KUKA KRL program: vw_bu_usr_s.src, vw_bu_usr_s.dat

--- vw_bu_usr_s.src ---
&ACCESS RV1
&COMMENT KS26
&REL 200
&PARAM DISKPATH = VW_User/Applikation/BU_Buersten
&PARAM TPUSER_VERSION = 8.3.0
DEF VW_BU_USR_S( )
;
;***************************************************
;*Technologiepaket Buersten                        *
;*                                                 *
;*Konzernstandard                                  *
;*Bearbeiter: C. Eisenknappl AUDI AG I/PG-C61      *
;*                                                 *
;* Aenderungsjournal:                              *
;*                                                 *
;***************************************************
;
END
;
;FOLD INIT BU
GLOBAL DEF BU_INIT( )
INT i
;
;FOLD Version Techpaket
Tech_BU.Name[]="KS26.01.002_20190612"
;ENDFOLD
;
;FOLD Vorbesetzung Meldungsausgabe
FOR i=1 TO 100
  n_BUS_Handle[i]=-1
  n_BUR_Handle[i]=-1
ENDFOR
;ENDFOLD
;
;FOLD BU BASE ADRESSEN INITIALISIEREN
BU_BASE_INIT( )
;ENDFOLD
;
END
;ENDFOLD
;
;***************************************************
;FOLD SAW BU
GLOBAL DEF BU_SAW( )
INT i
;
;
END
;ENDFOLD
;
;***************************************************
;FOLD RESET BU
GLOBAL DEF BU_RESET( )
INT i
;
;
END
;ENDFOLD
;
;***************************************************
;FOLD CANCEL BU
GLOBAL DEF BU_CANCEL( )
INT i
;
;
END
;ENDFOLD
;
;***************************************************
;FOLD LOOP BU
GLOBAL DEF BU_LOOP( )
BOOL bRet
;
;FOLD BU BASE ADRESSEN INITIALISIEREN
BU_BASE_INIT( )
;ENDFOLD
;
IF (BU_BASE_SL==HM_BASE_SL) THEN
  BU_Msg(1,#StateMsg)
ELSE
  IF (n_BUS_Handle[1]>-1) THEN
    bRet=Clear_KrlMsg(n_BUS_Handle[1])
    n_BUS_Handle[1]=-1
  ENDIF
ENDIF
;
IF ($EXT==TRUE) THEN
  $OUT[O_ACF_Teach]=FALSE
ENDIF
;
;ACF ohne Kraft
IF $IN[BU_BASE_SL+I_ACF_oh_Kra] THEN
  $OUT[O_ACF_oh_Kra]=TRUE
ELSE
  $OUT[O_ACF_oh_Kra]=FALSE
ENDIF
;
;ACF BA-Hand
IF $OUT[O_R_Hand] AND (NOT $COULD_START_MOTION) THEN
  $OUT[O_ACF_R_Hand]=TRUE
  $OUT[O_ACF_R_Auto]=FALSE
ENDIF
;
;ACF BA-AUTO
IF $OUT[O_R_Hand] AND ($OUT[O_R_Proz_akt] OR $OUT[O_R_bewegt]) OR $OUT[O_R_Auto] THEN
  $OUT[O_ACF_R_Hand]=FALSE
  $OUT[O_ACF_R_Auto]=TRUE
ENDIF
;
;Visualisierung config.mon
IF (ACF110==TRUE) THEN
  ACF_max_WEG=355
ENDIF
IF (ACF111==TRUE) THEN
  ACF_max_WEG=355
ENDIF
IF (ACF12x==TRUE) THEN
  ACF_max_WEG=480
ENDIF
IF (ACF131==TRUE) THEN
  ACF_max_WEG=480
ENDIF
ACF_Result_5=((SI_ACF_Istpos-ACF_max_WEG)*(-0.1))
IF NOT $IN[ACF_istneg] THEN
  ACF_istkraft_Hilf=SI_ACF_IstKraft
ELSE
  ACF_istkraft_Hilf=(SI_ACF_IstKraft*(-1))
ENDIF
ACF_Result_6=ACF_istkraft_Hilf
;
;Fehler Reset
IF NOT $COULD_START_MOTION THEN
  Timer_BUFeh=$ROB_TIMER
  BU_AutoReset=TRUE
ENDIF
IF ((BU_AutoReset==TRUE) AND NOT $IN[I_ACF_Sammel]) THEN
  BU_AutoReset=FALSE
ENDIF
$OUT[O_ACF_Reset]=(NOT $IN[I_ACF_Sammel] AND ($IN[I_R_Quit_St] OR $IN[I_R_Quit_Wei]) OR ($OUT[O_R_PERI_RDY] AND (BU_AutoReset==TRUE) AND (($ROB_TIMER-Timer_BUFeh)<1000)))
;
;BU Antriebe EIN
$OUT[O_BU_ANT_EIN]=$FLAG[F_BU_EIN] AND $FLAG[F_FB_PSPS] AND $OUT[O_R_Proz_akt] AND NOT $FLAG[F_o_Proz_SStep] AND NOT $FLAG[F_o_Proz_BMS] AND NOT $IN[I_FT_o_BT]
;
;Ausgabe Statusmeldungen an BMS
;Prozess aktiv
$OUT[BU_BASE_SL+O_BU_Proz_aktiv]=$OUT[O_R_Auto] AND $COULD_START_MOTION AND ($IN[I_BU_Proz_aktiv] OR (Messen_aktiv==TRUE))
;Messen aktiv
$OUT[BU_BASE_SL+O_BU_Messen_aktiv]=$OUT[O_R_Auto] AND $COULD_START_MOTION AND (Messen_aktiv==TRUE)
;Messfehler
$OUT[BU_BASE_SL+O_BU_Messfehler]=$OUT[O_R_Auto] AND $COULD_START_MOTION AND (Messfehler==TRUE)
;Sammelstoerung
$OUT[BU_BASE_SL+O_BU_Sammel]=$OUT[O_R_Auto] AND $COULD_START_MOTION AND NOT $IN[I_BU_Sammel]
;
ACF_ZCode=1
;
L_Bit_ACF(1)
;
END
;ENDFOLD
;
;***************************************************
;FOLD Lebensbit_ACF
DEF L_Bit_ACF(ACFNr:IN)
INT ACFNr,RobTimer
BOOL LBitACF,LBitFault,ErrLBit,bRet
;
ErrLBit = FALSE
LBitFault=FALSE
;
;Setzen / Rueksetzen Lebensbit Roboter
$OUT[O_ACF_LBit]=NOT $IN[I_ACF_LBit]
RobTimer=$ROB_TIMER
IF $IN[I_ACF_LBit]<>LBitState[ACFNr] THEN
  LBitTimeCnt[ACFNr]=RobTimer
ENDIF
IF ((RobTimer-LBitTimeCnt[ACFNr])>5000) THEN
  ErrLBit=TRUE
  ACF_LBitFeh[ACFNr]=TRUE
ENDIF
LBitState[ACFNr]=$IN[I_ACF_LBit]
IF ErrLBit THEN
  BU_Msg(2,#StateMsg)
ELSE
  IF (n_BUS_Handle[2]>-1) THEN
    bRet=Clear_KrlMsg(n_BUS_Handle[2])
    n_BUS_Handle[1]=-1
  ENDIF
  ACF_LBitFeh[ACFNr]=FALSE
ENDIF
;
END
;ENDFOLD
;
;***************************************************
;FOLD BU_BASE_INIT
DEF BU_BASE_INIT()
INT BaseResult
;
;BU SLAVE ADRESSIERUNG
BaseResult=BaseCheck(CF_BU_BASE_SL)
IF (BaseResult<>0) THEN
  CF_BU_BASE_SL=HM_BASE_SL
  BU_BASE_SL=HM_BASE_SL
ELSE
  BU_BASE_SL=CF_BU_BASE_SL
ENDIF
;
END
;ENDFOLD (BU_BASE_INIT)
;
;***************************************************
;FOLD BU_Meldungen
DEF BU_Msg(msg_nr:IN,MsgTyp:IN,BUNr:IN)
INT msg_nr, BUNr, Answer
DECL BUS_MsgType MsgTyp
DECL KrlMsg_T USER_MSG
DECL KrlMsgPar_T Par[3]
DECL KrlMsgOpt_T Opt
;
USER_MSG = { Modul[] "BU_S_Msg", Nr -1, Msg_txt[] " "}
Opt = { VL_Stop FALSE, Clear_P_Reset TRUE, Log_To_DB TRUE }
Par[1] = { Par_type #Value, Par_txt[] " " }
;
IF Varstate("BUNr")==#initialized then
  SWITCH BUNr
    CASE 1
      Par[1] = { Par_type #Value, Par_int 1 }
    CASE 2
      Par[1] = { Par_type #Value, Par_int 2 }
    CASE 3
      Par[1] = { Par_type #Value, Par_int 3 }
    CASE 4
      Par[1] = { Par_type #Value, Par_int 4 }
    CASE 5
      Par[1] = { Par_type #Value, Par_int 5 }
    CASE 6
      Par[1] = { Par_type #Value, Par_int 6 }
    DEFAULT
      Par[1] = { Par_type #Value, Par_txt[] " " }
  ENDSWITCH
ELSE
  Par[1] = { Par_type #Value, Par_txt[] " " }
ENDIF
;
IF ((n_BUS_Handle[msg_nr]<0) OR (MsgTyp==#NotifyMsg) OR (MsgTyp==#QuitMsg)) THEN
  USER_MSG.Nr = msg_nr
  SWITCH msg_nr
    CASE 1
	   USER_MSG.MSG_TXT[]="BU: Slave Startadresse ungueltig"
    CASE 2
	   USER_MSG.MSG_TXT[]="ACF: Keine Antwort auf Lebensbit"
    CASE 3
	   USER_MSG.MSG_TXT[]=" "
    CASE 4
	   USER_MSG.MSG_TXT[]=" "
    DEFAULT
	   USER_MSG.MSG_TXT[]="unbekannte Meldung"
  ENDSWITCH
  SWITCH MsgTyp
    CASE #StateMsg
      n_BUS_Handle[msg_nr] = Set_KrlMsg (#State, USER_MSG, Par[], Opt) ;Ausgabe Statusmeldung
    CASE #QuitMsg
      n_BUS_Handle[msg_nr] = Set_KrlMsg (#Quit, USER_MSG, Par[], Opt) ;Ausgabe Quittierungsmeldung
    CASE #NotifyMsg
      n_BUS_Handle[msg_nr] = Set_KrlMsg (#Notify, USER_MSG, Par[], Opt) ;Ausgabe Hinweismeldung
    DEFAULT
      n_BUS_Handle[msg_nr] = Set_KrlMsg (#Quit, USER_MSG, Par[], Opt) ;Ausgabe Quittierungsmeldung
  ENDSWITCH
ENDIF
END
;
;ENDFOLD (BU Meldungen)

--- vw_bu_usr_s.dat ---
&ACCESS  RV
&COMMENT KS26
&PARAM DISKPATH = VW_User/Applikation/BU_Buersten
&PARAM TPUSER_VERSION = 8.3.0
&REL 200
DEFDAT  vw_bu_usr_s PUBLIC
;
;***************************************************
;*Technologiepaket Buersten                        *
;*                                                 *
;*Konzernstandard                                  *
;*Bearbeiter: C. Eisenknappl AUDI AG I/PG-C61      *
;*                                                 *
;* Erstellt am:                                    *
;* 2014.09.25 CE                                   *
;*                                                 *
;* 2015.01.08 LE  Vorb. Meldungsausg im INIT entf. *
;***************************************************
;
;Tech_Version
STRUC _Tech_BU CHAR Name[20],INT Datum
DECL _Tech_BU Tech_BU
;
;BU
;VARIABLEN INTEGER
GLOBAL INT BU_Result=0
GLOBAL INT BU_Schwellwert=140
GLOBAL INT BU_Erhoehung=160
GLOBAL INT TOOL_NR=0
GLOBAL INT Default_BU_BASE_SL=193
GLOBAL INT CF_BU_BASE_SL=449
GLOBAL INT CF_ACF_BASE_SL=449
GLOBAL INT Timer_BUFeh=0
;VARIABLEN REAL
GLOBAL REAL MESS_P_Z=0.0
GLOBAL REAL DELTA_Z=0.0
GLOBAL REAL DELTA=0.0
GLOBAL REAL BU_Verschleiss=0.0
GLOBAL REAL SUCH_WEG=0.0
GLOBAL REAL SUCH_VEL=0.01000000 ;max. Suchgeschwindigkeit [m/s]
;VARIABLEN BOOL
GLOBAL BOOL MIT_BU=FALSE
GLOBAL BOOL Messen_aktiv=FALSE
GLOBAL BOOL Messfehler=FALSE
GLOBAL BOOL Referenzfahrt=FALSE
GLOBAL BOOL BU_AutoReset=FALSE
;FLAGS
GLOBAL INT F_BU_EIN=620
GLOBAL INT F_BU_IBN=621
;BU SLAVE ADRESSIERUNG
GLOBAL INT BU_BASE_SL=449 ;BU Indirekte Slave Adressen
;Slave Eingaenge
GLOBAL INT I_BU_o_Proz=0
;Slave Ausgaenge
GLOBAL INT O_BU_Proz_aktiv=0
GLOBAL INT O_BU_Messen_aktiv=1
GLOBAL INT O_BU_Vw_Standmenge=2
GLOBAL INT O_BU_max_Standmenge=3
GLOBAL INT O_BU_Messfehler=5
GLOBAL INT O_BU_Stoer=6
GLOBAL INT O_BU_Sammel=7
;Master Eingaenge
GLOBAL INT I_BU_Proz_aktiv=2952
GLOBAL INT I_BU_Sammel=2960
;Master Ausgaenge
GLOBAL INT O_BU_ANT_EIN=2952
;
;ACF
;VARIABLEN REAL
GLOBAL REAL ACF_Result_1=0.0
GLOBAL REAL ACF_Result_2=0.0
GLOBAL REAL ACF_Result_3=0.0
GLOBAL REAL ACF_Result_4=0.0
GLOBAL REAL ACF_Result_5=0.0
GLOBAL REAL ACF_Result_6=0.0
GLOBAL REAL ACF_istkraft_Hilf=0.0
;VARIABLEN BOOL
GLOBAL BOOL MIT_ACF=FALSE
GLOBAL BOOL ACF110=FALSE
GLOBAL BOOL ACF111=FALSE
GLOBAL BOOL ACF12x=FALSE
GLOBAL BOOL ACF131=FALSE
;VARIABLEN INTEGER
GLOBAL INT ACF_max_WEG=0
;Slave Eingaenge
GLOBAL INT I_ACF_oh_Kra=1
;Master Eingaenge
GLOBAL INT I_ACF_LBit=2947
GLOBAL INT I_ACF_R_Hand=2949
GLOBAL INT I_ACF_R_Auto=2950
GLOBAL INT I_ACF_teach=2951
GLOBAL INT I_ACF_Kontakt=2953
GLOBAL INT ACF_istneg=2976
GLOBAL INT I_ACF_Sammel=2960
;Master Ausgaenge
GLOBAL INT O_ACF_Reset=2945
GLOBAL INT O_ACF_oh_Kra=2946
GLOBAL INT O_ACF_Teach=2951
GLOBAL INT O_ACF_LBit=2947
GLOBAL INT O_ACF_R_Hand=2949
GLOBAL INT O_ACF_R_Auto=2950
;
SIGNAL SI_ACF_Istpos $IN[2977]  TO $IN[2992]
SIGNAL SI_ACF_IstKraft $IN[2961]  TO $IN[2975]
SIGNAL ACF_ZCode $OUT[2957]  TO $OUT[2959]
;
;Lebensbit ACF
BOOL LBitState[2]
LBitState[1]=FALSE
LBitState[2]=FALSE
BOOL ACF_LBitFeh[2]
ACF_LBitFeh[1]=FALSE
ACF_LBitFeh[2]=FALSE
;
INT LBitTimeCnt[2]
LBitTimeCnt[1]=-1
LBitTimeCnt[2]=-1
INT ErrACFNr=-1
;
;Meldungsausgabe
ENUM BUS_MsgType StateMsg,QuitMsg,NotifyMsg
GLOBAL INT n_BUS_Handle[100]
GLOBAL INT n_BUR_Handle[100]
INT nMsgNum=0
INT RemMsgNum=0
;
ENDDAT
